ABB RobotStudio station: Device-1.rspag

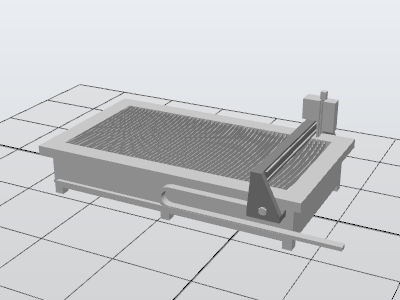
Station Device (saved by RobotStudio 24.1.10713.1)
Layout (positions relative to the parent item):
  - Device [mechanism, from Module 3\Device.rslib] at (0, 0, 0) mm; joint values [-0.65, 0.25, -0.0886] (rad or m)
